// TIA Portal V16 export
// export: Created 2024-09-05T17:39:22.8012571Z, ExportSetting WithDefaults, DisplayName Totally Integrated Automation Portal, DisplayVersion V16 Update 6, DisplayName TIA Portal Version Control Interface, DisplayVersion V16 Update 2, DisplayName TIA Portal Openness, DisplayVersion V16 Update 6, DisplayName STEP 7 Professional, DisplayVersion V16 Update 6, DisplayName STEP 7 Safety, DisplayVersion V16, DisplayName WinCC Advanced, DisplayVersion V16 Update 6
FUNCTION_BLOCK "IJCoreMain"   // FB1000, LAD
TITLE = IJCore Main
{ S7_Optimized_Access := 'TRUE' }
VERSION : 0.1
// stored: AutoNumber false, IsIECCheckEnabled false, IsRetainMemResEnabled false, MemoryReserve 100, SetENOAutomatically false, UDAEnableTagReadback false
   VAR
      Enable : Bool;
      Mode : UInt;
      Indicator : Int;
      AlarmReset : Bool;
      AWAKE_SIGNAL { S7_SetPoint := 'True'} : "AWAKE_SIGNAL";
      MSG : Array[1..20] of "IJCoreMessageProcotol";
      NFP { S7_SetPoint := 'True'} : Array[1..4] of String[30];
   END_VAR
   VAR_TEMP
      MessageDone : Bool;
      Answer : DInt;
      Fault : DInt;
   END_VAR
   VAR CONSTANT
      STA : Int := 5;
      CNF : Int := 1;
      TRC : Int := 13;
      PFC : Int := 9;
      TRR : Int := 7;
   END_VAR
BEGIN

REGION Network 1
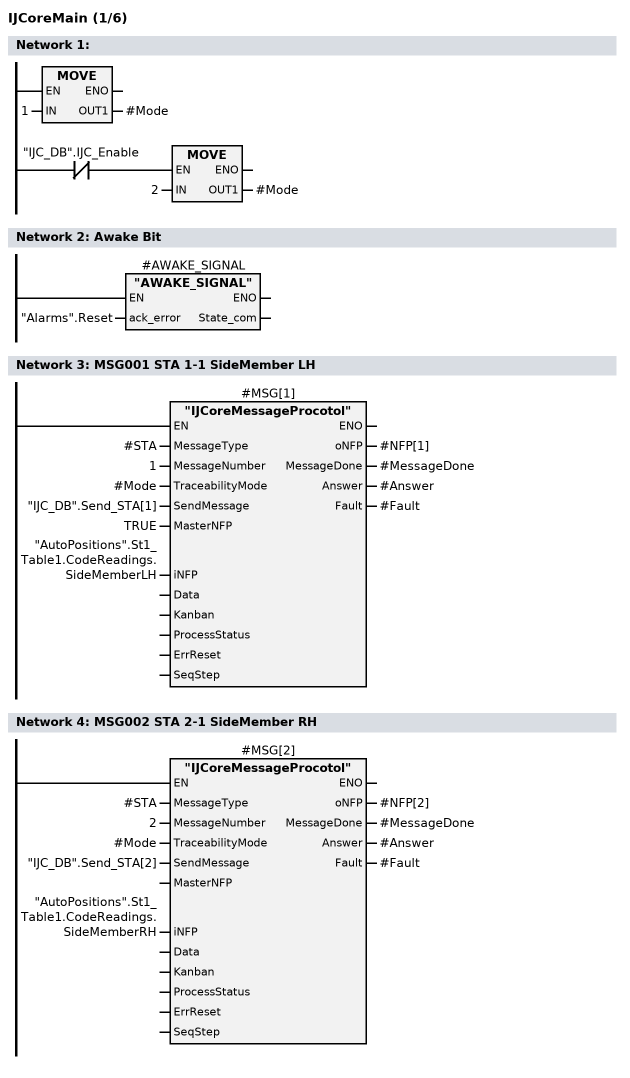
   RUNG wire#powerrail
      Move(in := 1, out1 => #Mode)
   END_RUNG
   RUNG wire#powerrail
      I_Contact( "IJC_DB".IJC_Enable )
      Move(in := 2, out1 => #Mode)
   END_RUNG
   // the same network as SCL:
   #Mode := 1;
   IF NOT "IJC_DB".IJC_Enable THEN #Mode := 2; END_IF;
END_REGION

REGION Network 2: Awake Bit
   RUNG wire#powerrail
      #AWAKE_SIGNAL(ack_error := "Alarms".Reset, State_com =>)
   END_RUNG
   // the same network as SCL:
   #AWAKE_SIGNAL(ack_error := "Alarms".Reset);   // "AWAKE_SIGNAL"
END_REGION

REGION Network 3: MSG001 STA 1-1 SideMember LH
   RUNG wire#powerrail
      #MSG[1](MessageType := #STA, MessageNumber := 1, TraceabilityMode := #Mode, SendMessage := "IJC_DB".Send_STA[1], MasterNFP := TRUE, iNFP := "AutoPositions".St1_Table1.CodeReadings.SideMemberLH, Data :=, Kanban :=, ProcessStatus :=, ErrReset :=, SeqStep :=, oNFP => #NFP[1], MessageDone => #MessageDone, Answer => #Answer, Fault => #Fault)
   END_RUNG
   // the same network as SCL:
   #MSG[1](MessageType := #STA,   // "IJCoreMessageProcotol"
           MessageNumber := 1,
           TraceabilityMode := #Mode,
           SendMessage := "IJC_DB".Send_STA[1],
           MasterNFP := TRUE,
           iNFP := "AutoPositions".St1_Table1.CodeReadings.SideMemberLH,
           oNFP => #NFP[1],
           MessageDone => #MessageDone,
           Answer => #Answer,
           Fault => #Fault);
END_REGION

REGION Network 4: MSG002 STA 2-1 SideMember RH
   RUNG wire#powerrail
      #MSG[2](MessageType := #STA, MessageNumber := 2, TraceabilityMode := #Mode, SendMessage := "IJC_DB".Send_STA[2], MasterNFP :=, iNFP := "AutoPositions".St1_Table1.CodeReadings.SideMemberRH, Data :=, Kanban :=, ProcessStatus :=, ErrReset :=, SeqStep :=, oNFP => #NFP[2], MessageDone => #MessageDone, Answer => #Answer, Fault => #Fault)
   END_RUNG
   // the same network as SCL:
   #MSG[2](MessageType := #STA,   // "IJCoreMessageProcotol"
           MessageNumber := 2,
           TraceabilityMode := #Mode,
           SendMessage := "IJC_DB".Send_STA[2],
           iNFP := "AutoPositions".St1_Table1.CodeReadings.SideMemberRH,
           oNFP => #NFP[2],
           MessageDone => #MessageDone,
           Answer => #Answer,
           Fault => #Fault);
END_REGION

REGION Network 5: MSG003 STA 3-1 Front Tube
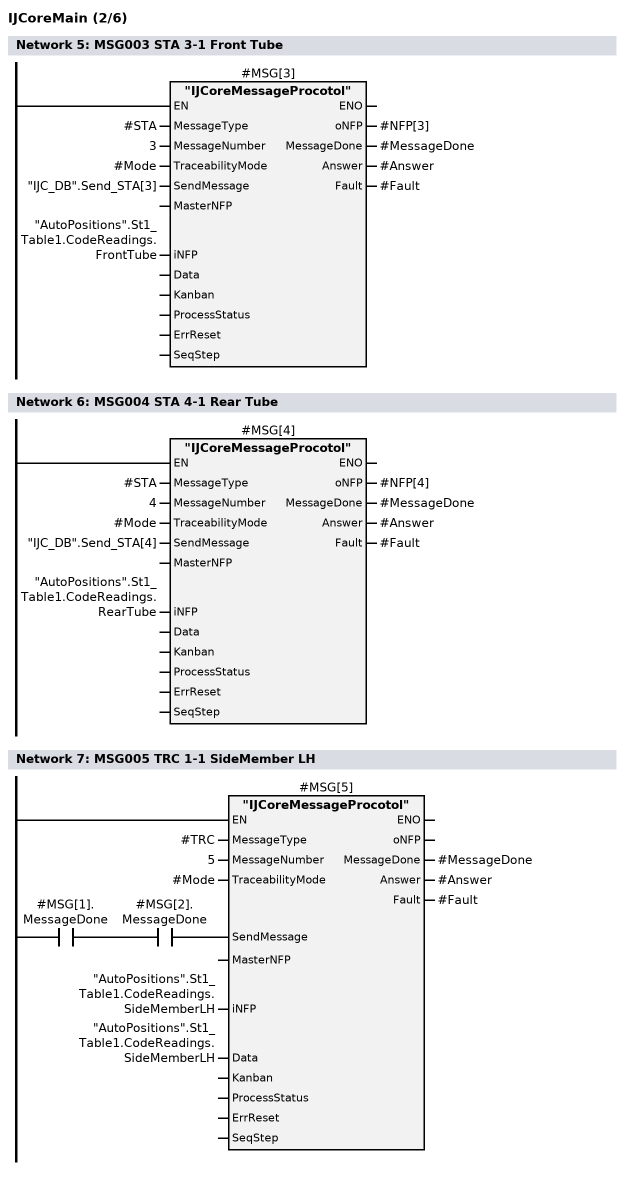
   RUNG wire#powerrail
      #MSG[3](MessageType := #STA, MessageNumber := 3, TraceabilityMode := #Mode, SendMessage := "IJC_DB".Send_STA[3], MasterNFP :=, iNFP := "AutoPositions".St1_Table1.CodeReadings.FrontTube, Data :=, Kanban :=, ProcessStatus :=, ErrReset :=, SeqStep :=, oNFP => #NFP[3], MessageDone => #MessageDone, Answer => #Answer, Fault => #Fault)
   END_RUNG
   // the same network as SCL:
   #MSG[3](MessageType := #STA,   // "IJCoreMessageProcotol"
           MessageNumber := 3,
           TraceabilityMode := #Mode,
           SendMessage := "IJC_DB".Send_STA[3],
           iNFP := "AutoPositions".St1_Table1.CodeReadings.FrontTube,
           oNFP => #NFP[3],
           MessageDone => #MessageDone,
           Answer => #Answer,
           Fault => #Fault);
END_REGION

REGION Network 6: MSG004 STA 4-1 Rear Tube
   RUNG wire#powerrail
      #MSG[4](MessageType := #STA, MessageNumber := 4, TraceabilityMode := #Mode, SendMessage := "IJC_DB".Send_STA[4], MasterNFP :=, iNFP := "AutoPositions".St1_Table1.CodeReadings.RearTube, Data :=, Kanban :=, ProcessStatus :=, ErrReset :=, SeqStep :=, oNFP => #NFP[4], MessageDone => #MessageDone, Answer => #Answer, Fault => #Fault)
   END_RUNG
   // the same network as SCL:
   #MSG[4](MessageType := #STA,   // "IJCoreMessageProcotol"
           MessageNumber := 4,
           TraceabilityMode := #Mode,
           SendMessage := "IJC_DB".Send_STA[4],
           iNFP := "AutoPositions".St1_Table1.CodeReadings.RearTube,
           oNFP => #NFP[4],
           MessageDone => #MessageDone,
           Answer => #Answer,
           Fault => #Fault);
END_REGION

REGION Network 7: MSG005 TRC 1-1 SideMember LH
   RUNG wire#powerrail
      #MSG[5](SendMessage := wire#w1, MessageType := #TRC, MessageNumber := 5, TraceabilityMode := #Mode, MasterNFP :=, iNFP := "AutoPositions".St1_Table1.CodeReadings.SideMemberLH, Data := "AutoPositions".St1_Table1.CodeReadings.SideMemberLH, Kanban :=, ProcessStatus :=, ErrReset :=, SeqStep :=, oNFP =>, MessageDone => #MessageDone, Answer => #Answer, Fault => #Fault)
   END_RUNG
   RUNG wire#powerrail
      Contact( #MSG[1].MessageDone )
      Contact( #MSG[2].MessageDone )
   END_RUNG wire#w1
   // the same network as SCL:
   #MSG[5](MessageType := #TRC,   // "IJCoreMessageProcotol"
           MessageNumber := 5,
           TraceabilityMode := #Mode,
           SendMessage := #MSG[1].MessageDone AND #MSG[2].MessageDone,
           iNFP := "AutoPositions".St1_Table1.CodeReadings.SideMemberLH,
           Data := "AutoPositions".St1_Table1.CodeReadings.SideMemberLH,
           MessageDone => #MessageDone,
           Answer => #Answer,
           Fault => #Fault);
END_REGION

REGION Network 8: MSG006 TRC 1-2 SideMember RH
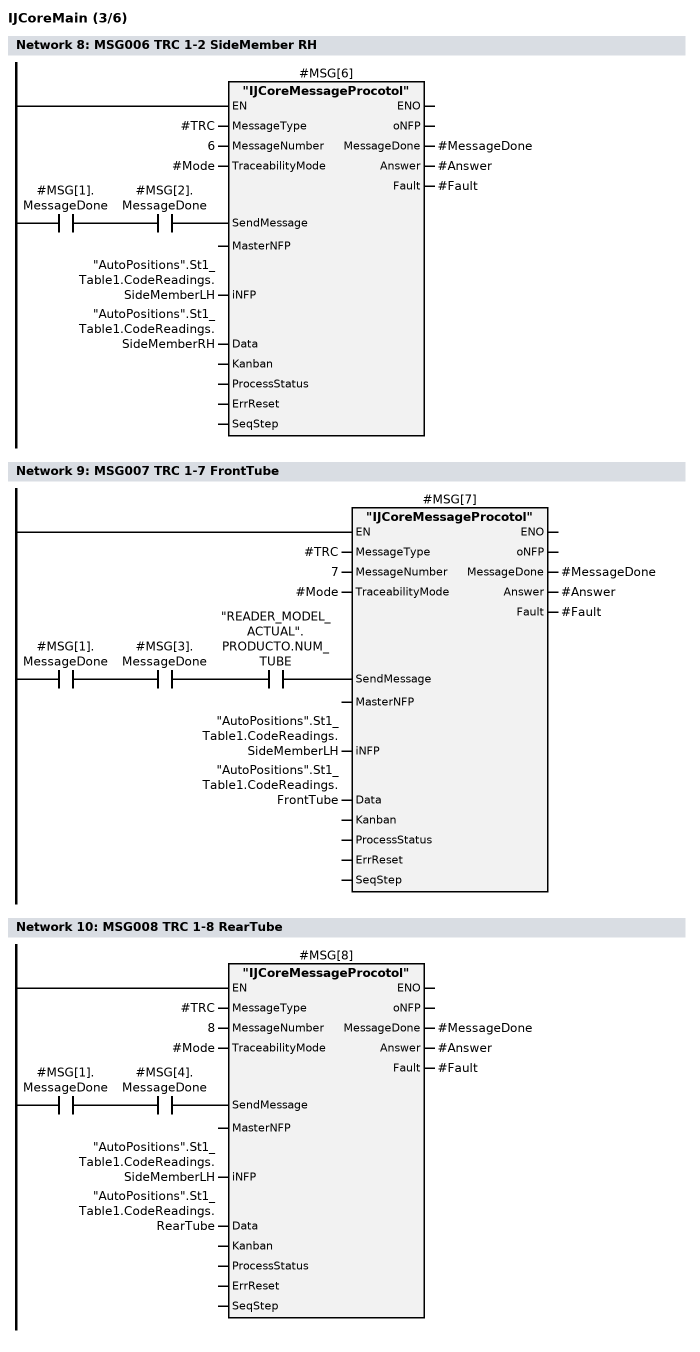
   RUNG wire#powerrail
      #MSG[6](SendMessage := wire#w1, MessageType := #TRC, MessageNumber := 6, TraceabilityMode := #Mode, MasterNFP :=, iNFP := "AutoPositions".St1_Table1.CodeReadings.SideMemberLH, Data := "AutoPositions".St1_Table1.CodeReadings.SideMemberRH, Kanban :=, ProcessStatus :=, ErrReset :=, SeqStep :=, oNFP =>, MessageDone => #MessageDone, Answer => #Answer, Fault => #Fault)
   END_RUNG
   RUNG wire#powerrail
      Contact( #MSG[1].MessageDone )
      Contact( #MSG[2].MessageDone )
   END_RUNG wire#w1
   // the same network as SCL:
   #MSG[6](MessageType := #TRC,   // "IJCoreMessageProcotol"
           MessageNumber := 6,
           TraceabilityMode := #Mode,
           SendMessage := #MSG[1].MessageDone AND #MSG[2].MessageDone,
           iNFP := "AutoPositions".St1_Table1.CodeReadings.SideMemberLH,
           Data := "AutoPositions".St1_Table1.CodeReadings.SideMemberRH,
           MessageDone => #MessageDone,
           Answer => #Answer,
           Fault => #Fault);
END_REGION

REGION Network 9: MSG007 TRC 1-7 FrontTube
   RUNG wire#powerrail
      #MSG[7](SendMessage := wire#w1, MessageType := #TRC, MessageNumber := 7, TraceabilityMode := #Mode, MasterNFP :=, iNFP := "AutoPositions".St1_Table1.CodeReadings.SideMemberLH, Data := "AutoPositions".St1_Table1.CodeReadings.FrontTube, Kanban :=, ProcessStatus :=, ErrReset :=, SeqStep :=, oNFP =>, MessageDone => #MessageDone, Answer => #Answer, Fault => #Fault)
   END_RUNG
   RUNG wire#powerrail
      Contact( #MSG[1].MessageDone )
      Contact( #MSG[3].MessageDone )
      Contact( "READER_MODEL_ACTUAL".PRODUCTO.NUM_TUBE )
   END_RUNG wire#w1
   // the same network as SCL:
   #MSG[7](MessageType := #TRC,   // "IJCoreMessageProcotol"
           MessageNumber := 7,
           TraceabilityMode := #Mode,
           SendMessage := #MSG[1].MessageDone AND #MSG[3].MessageDone AND "READER_MODEL_ACTUAL".PRODUCTO.NUM_TUBE,
           iNFP := "AutoPositions".St1_Table1.CodeReadings.SideMemberLH,
           Data := "AutoPositions".St1_Table1.CodeReadings.FrontTube,
           MessageDone => #MessageDone,
           Answer => #Answer,
           Fault => #Fault);
END_REGION

REGION Network 10: MSG008 TRC 1-8 RearTube
   RUNG wire#powerrail
      #MSG[8](SendMessage := wire#w1, MessageType := #TRC, MessageNumber := 8, TraceabilityMode := #Mode, MasterNFP :=, iNFP := "AutoPositions".St1_Table1.CodeReadings.SideMemberLH, Data := "AutoPositions".St1_Table1.CodeReadings.RearTube, Kanban :=, ProcessStatus :=, ErrReset :=, SeqStep :=, oNFP =>, MessageDone => #MessageDone, Answer => #Answer, Fault => #Fault)
   END_RUNG
   RUNG wire#powerrail
      Contact( #MSG[1].MessageDone )
      Contact( #MSG[4].MessageDone )
   END_RUNG wire#w1
   // the same network as SCL:
   #MSG[8](MessageType := #TRC,   // "IJCoreMessageProcotol"
           MessageNumber := 8,
           TraceabilityMode := #Mode,
           SendMessage := #MSG[1].MessageDone AND #MSG[4].MessageDone,
           iNFP := "AutoPositions".St1_Table1.CodeReadings.SideMemberLH,
           Data := "AutoPositions".St1_Table1.CodeReadings.RearTube,
           MessageDone => #MessageDone,
           Answer => #Answer,
           Fault => #Fault);
END_REGION

REGION Network 11: MSG009 TRR 1-1 Results of riveting
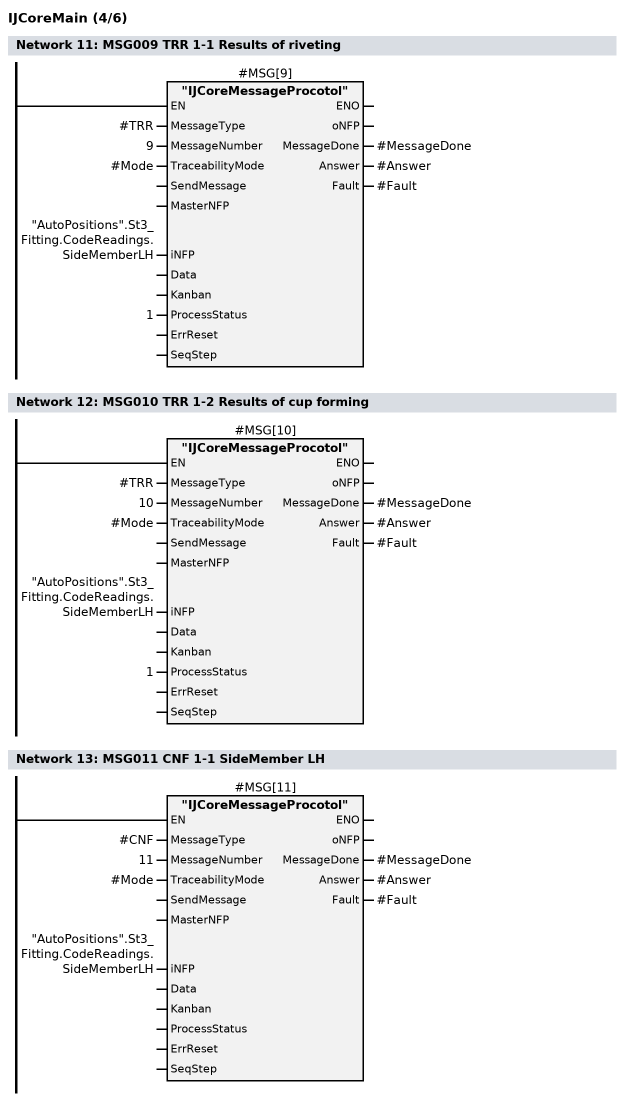
   RUNG wire#powerrail
      #MSG[9](MessageType := #TRR, MessageNumber := 9, TraceabilityMode := #Mode, SendMessage :=, MasterNFP :=, iNFP := "AutoPositions".St3_Fitting.CodeReadings.SideMemberLH, Data :=, Kanban :=, ProcessStatus := 1, ErrReset :=, SeqStep :=, oNFP =>, MessageDone => #MessageDone, Answer => #Answer, Fault => #Fault)
   END_RUNG
   // the same network as SCL:
   #MSG[9](MessageType := #TRR,   // "IJCoreMessageProcotol"
           MessageNumber := 9,
           TraceabilityMode := #Mode,
           iNFP := "AutoPositions".St3_Fitting.CodeReadings.SideMemberLH,
           ProcessStatus := 1,
           MessageDone => #MessageDone,
           Answer => #Answer,
           Fault => #Fault);
END_REGION

REGION Network 12: MSG010 TRR 1-2 Results of cup forming
   RUNG wire#powerrail
      #MSG[10](MessageType := #TRR, MessageNumber := 10, TraceabilityMode := #Mode, SendMessage :=, MasterNFP :=, iNFP := "AutoPositions".St3_Fitting.CodeReadings.SideMemberLH, Data :=, Kanban :=, ProcessStatus := 1, ErrReset :=, SeqStep :=, oNFP =>, MessageDone => #MessageDone, Answer => #Answer, Fault => #Fault)
   END_RUNG
   // the same network as SCL:
   #MSG[10](MessageType := #TRR,   // "IJCoreMessageProcotol"
            MessageNumber := 10,
            TraceabilityMode := #Mode,
            iNFP := "AutoPositions".St3_Fitting.CodeReadings.SideMemberLH,
            ProcessStatus := 1,
            MessageDone => #MessageDone,
            Answer => #Answer,
            Fault => #Fault);
END_REGION

REGION Network 13: MSG011 CNF 1-1 SideMember LH
   RUNG wire#powerrail
      #MSG[11](MessageType := #CNF, MessageNumber := 11, TraceabilityMode := #Mode, SendMessage :=, MasterNFP :=, iNFP := "AutoPositions".St3_Fitting.CodeReadings.SideMemberLH, Data :=, Kanban :=, ProcessStatus :=, ErrReset :=, SeqStep :=, oNFP =>, MessageDone => #MessageDone, Answer => #Answer, Fault => #Fault)
   END_RUNG
   // the same network as SCL:
   #MSG[11](MessageType := #CNF,   // "IJCoreMessageProcotol"
            MessageNumber := 11,
            TraceabilityMode := #Mode,
            iNFP := "AutoPositions".St3_Fitting.CodeReadings.SideMemberLH,
            MessageDone => #MessageDone,
            Answer => #Answer,
            Fault => #Fault);
END_REGION

REGION Network 14: MSG012 CNF 1-2 SideMember RH
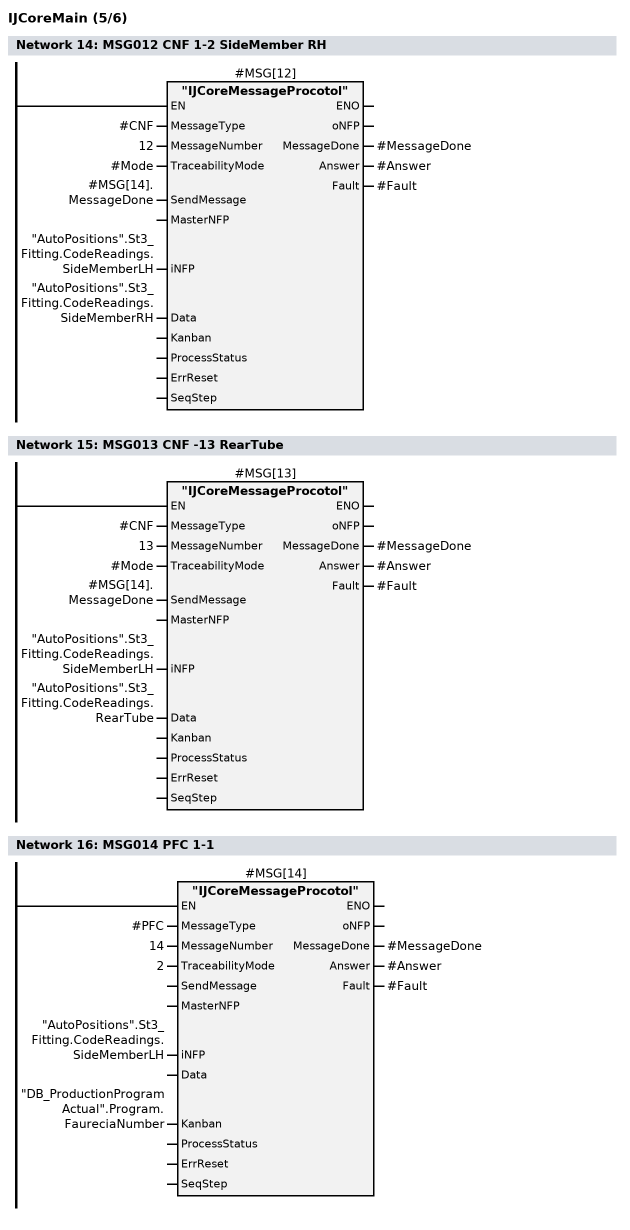
   RUNG wire#powerrail
      #MSG[12](MessageType := #CNF, MessageNumber := 12, TraceabilityMode := #Mode, SendMessage := #MSG[14].MessageDone, MasterNFP :=, iNFP := "AutoPositions".St3_Fitting.CodeReadings.SideMemberLH, Data := "AutoPositions".St3_Fitting.CodeReadings.SideMemberRH, Kanban :=, ProcessStatus :=, ErrReset :=, SeqStep :=, oNFP =>, MessageDone => #MessageDone, Answer => #Answer, Fault => #Fault)
   END_RUNG
   // the same network as SCL:
   #MSG[12](MessageType := #CNF,   // "IJCoreMessageProcotol"
            MessageNumber := 12,
            TraceabilityMode := #Mode,
            SendMessage := #MSG[14].MessageDone,
            iNFP := "AutoPositions".St3_Fitting.CodeReadings.SideMemberLH,
            Data := "AutoPositions".St3_Fitting.CodeReadings.SideMemberRH,
            MessageDone => #MessageDone,
            Answer => #Answer,
            Fault => #Fault);
END_REGION

REGION Network 15: MSG013 CNF -13 RearTube
   RUNG wire#powerrail
      #MSG[13](MessageType := #CNF, MessageNumber := 13, TraceabilityMode := #Mode, SendMessage := #MSG[14].MessageDone, MasterNFP :=, iNFP := "AutoPositions".St3_Fitting.CodeReadings.SideMemberLH, Data := "AutoPositions".St3_Fitting.CodeReadings.RearTube, Kanban :=, ProcessStatus :=, ErrReset :=, SeqStep :=, oNFP =>, MessageDone => #MessageDone, Answer => #Answer, Fault => #Fault)
   END_RUNG
   // the same network as SCL:
   #MSG[13](MessageType := #CNF,   // "IJCoreMessageProcotol"
            MessageNumber := 13,
            TraceabilityMode := #Mode,
            SendMessage := #MSG[14].MessageDone,
            iNFP := "AutoPositions".St3_Fitting.CodeReadings.SideMemberLH,
            Data := "AutoPositions".St3_Fitting.CodeReadings.RearTube,
            MessageDone => #MessageDone,
            Answer => #Answer,
            Fault => #Fault);
END_REGION

REGION Network 16: MSG014 PFC 1-1
   RUNG wire#powerrail
      #MSG[14](MessageType := #PFC, MessageNumber := 14, TraceabilityMode := 2, SendMessage :=, MasterNFP :=, iNFP := "AutoPositions".St3_Fitting.CodeReadings.SideMemberLH, Data :=, Kanban := "DB_ProductionProgramActual".Program.FaureciaNumber, ProcessStatus :=, ErrReset :=, SeqStep :=, oNFP =>, MessageDone => #MessageDone, Answer => #Answer, Fault => #Fault)
   END_RUNG
   // the same network as SCL:
   #MSG[14](MessageType := #PFC,   // "IJCoreMessageProcotol"
            MessageNumber := 14,
            TraceabilityMode := 2,
            iNFP := "AutoPositions".St3_Fitting.CodeReadings.SideMemberLH,
            Kanban := "DB_ProductionProgramActual".Program.FaureciaNumber,
            MessageDone => #MessageDone,
            Answer => #Answer,
            Fault => #Fault);
END_REGION

REGION Network 17: MSG015 CNF 1-4 Front Tube
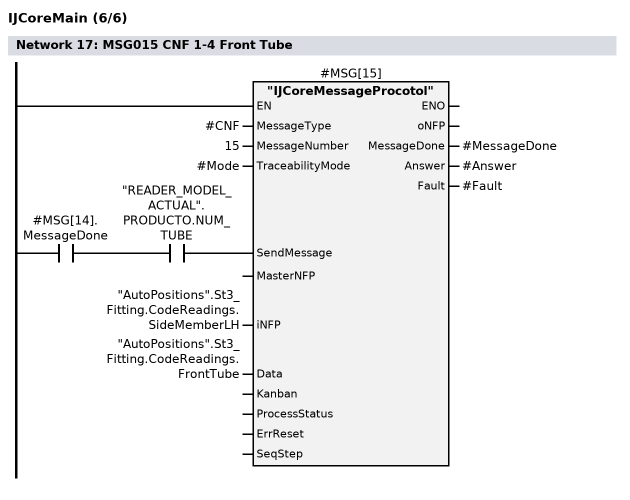
   RUNG wire#powerrail
      #MSG[15](SendMessage := wire#w1, MessageType := #CNF, MessageNumber := 15, TraceabilityMode := #Mode, MasterNFP :=, iNFP := "AutoPositions".St3_Fitting.CodeReadings.SideMemberLH, Data := "AutoPositions".St3_Fitting.CodeReadings.FrontTube, Kanban :=, ProcessStatus :=, ErrReset :=, SeqStep :=, oNFP =>, MessageDone => #MessageDone, Answer => #Answer, Fault => #Fault)
   END_RUNG
   RUNG wire#powerrail
      Contact( #MSG[14].MessageDone )
      Contact( "READER_MODEL_ACTUAL".PRODUCTO.NUM_TUBE )
   END_RUNG wire#w1
   // the same network as SCL:
   #MSG[15](MessageType := #CNF,   // "IJCoreMessageProcotol"
            MessageNumber := 15,
            TraceabilityMode := #Mode,
            SendMessage := #MSG[14].MessageDone AND "READER_MODEL_ACTUAL".PRODUCTO.NUM_TUBE,
            iNFP := "AutoPositions".St3_Fitting.CodeReadings.SideMemberLH,
            Data := "AutoPositions".St3_Fitting.CodeReadings.FrontTube,
            MessageDone => #MessageDone,
            Answer => #Answer,
            Fault => #Fault);
END_REGION
END_FUNCTION_BLOCK
